// TIA Portal V18 export
FUNCTION "01_Settings" : Void   // FC2, F_FBD
{ S7_Optimized_Access := 'TRUE' }
BEGIN

REGION Network 1: To be used in case of overall settings
   // for example in case of Tristate diagnostic
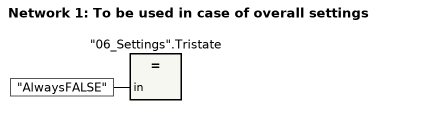
   "06_Settings".Tristate := "AlwaysFALSE";
END_REGION
END_FUNCTION
